(* PLC project Unnamed, Unknown Unnamed 1 *)
(* stored: creationDateTime 2026-03-25T00:31:42, modificationDateTime 2026-03-25T00:31:42 *)

PROGRAM main
  VAR
    PB1 AT %IX0.0 : BOOL;  (* 푸시버튼 (입력) *)
    LED AT %QX0.1 : BOOL;  (* 푸시버튼 (입력) *)
  END_VAR
  VAR
    T1 : TON;  (* 아두이노 내장 LED (출력) *)
    Blink_State : BOOL;  (* 현재 깜빡임 상태 저장 *)
  END_VAR

            (* 1초 타이머 설정 *)
T1(IN := NOT T1.Q, PT := T#1s);

(* 타이머가 완료될 때마다 LED 상태를 반전 *)
IF T1.Q THEN
    Blink_State := NOT Blink_State;
END_IF;

(* 최종 출력을 LED에 전달 *)
LED := Blink_State;

          
END_PROGRAM

CONFIGURATION Config0
  RESOURCE Res0 ON PLC
    TASK task0(INTERVAL := T#20ms, PRIORITY := 1);
    PROGRAM instance0 WITH task0 : main;
  END_RESOURCE
END_CONFIGURATION
